{attribute 'GeneratedUsingTerminal: AT2020-0250-0019'}
{attribute addProperty BoxType "AT2020-0250-0019"}
{attribute addProperty Id "A_0085_AT2050_5500_0018_AT2050_5500AT2050_33A3DF1B80"}
{attribute addProperty CRC "703496822"}
{attribute addProperty Size "80"}
TYPE A_0060_AT2020_0250_0019_AT2020_0250_29EE8276 EXTENDS AT2020_2EA6C9BF :
STRUCT
	{attribute addProperty Name "A_0085_AT2050_5500_0018_AT2050_5500"}
	{attribute addProperty PreviousPort "A_0060(AT2020-0250-0019) (AT2020-0250) : B"}
	A_0085_AT2050_5500_0018_AT2050_5500 : AT2050_33A3DF1B;
END_STRUCT
END_TYPE

(* stored: Version 1.2.0.0, ProductVersion 3.1.4024.9
   DUT A_0060_AT2020_0250_0019_AT2020_0250_29EE8276: Id {897eca45-246e-4f44-824e-28f0f68bbe80} *)
